# EPICS autosave request: CARSApp/Db/FluorTomo.req
$(P)$(Q):CountTime
$(P)$(Q):NFrames
$(P)$(Q):Request
$(P)$(Q):host
$(P)$(Q):dir
$(P)$(Q):subdir
$(P)$(Q):filebase
$(P)$(Q):format
$(P)$(Q):fileext
$(P)$(Q):TSTAMP
$(P)$(Q):UNIXTS
